INTERFACE I_Telescope

PROPERTY Altitude : LREAL
GET
END_GET
END_PROPERTY

PROPERTY Azimuth : LREAL
GET
END_GET
END_PROPERTY

PROPERTY CoverAutoOpen : BOOL
GET
END_GET
SET
END_SET
END_PROPERTY

PROPERTY Declination : LREAL
GET
END_GET
END_PROPERTY

METHOD ABSTRACT Home : BOOL
VAR_INPUT
END_VAR
END_METHOD

METHOD Init : BOOL
VAR_INPUT
END_VAR
END_METHOD

METHOD ABSTRACT Park : BOOL
VAR_INPUT
END_VAR
END_METHOD

METHOD Reset : BOOL
VAR_INPUT
END_VAR
END_METHOD

PROPERTY RightAscension : LREAL
GET
END_GET
END_PROPERTY

METHOD Slew : BOOL
VAR_INPUT
	fAzimuth		: LREAL;
	fAltitude		: LREAL;
END_VAR
END_METHOD

METHOD Stop : BOOL
VAR_INPUT
END_VAR
END_METHOD

METHOD Track : BOOL
VAR_INPUT
	fRightAscension	: LREAL;
	fDeclination	: LREAL;
END_VAR
END_METHOD

END_INTERFACE

(* stored: Version 1.1.0.1, ProductVersion 3.1.4024.15
   Itf I_Telescope: Id {5003d6e3-4b52-4cb8-a028-b0ab2a6b3370}
   Property Altitude: Id {ce60f76f-3a5f-482f-9275-0897e7d29930}
   Get Get: Id {58c7dbd3-1bf7-4cb4-96b8-f33be68a1ee1}
   Property Azimuth: Id {32bf6858-c17f-4c7b-8e70-4ffdf9df410d}
   Get Get: Id {63e5582f-b70a-403e-801b-c0e6f9154192}
   Property CoverAutoOpen: Id {f8160a73-8302-45f4-9c7c-d48b30d350e4}
   Get Get: Id {d18e5bdf-2192-4bf0-9513-4be35621818a}
   Set Set: Id {292bc5f3-fb7f-4633-b013-091fb338acaf}
   Property Declination: Id {a5cf9f3f-1ec9-4cca-8bd9-8121481b9a9f}
   Get Get: Id {fcb6c1b5-27f0-4565-aed9-45fc0ce88d7e}
   Method Home: Id {2fc689c7-e332-49bc-87f2-069b41e58195}
   Method Init: Id {a446f50b-d891-42c3-bcd4-e100ad4f506e}
   Method Park: Id {4989c55f-52d0-4389-8fa2-916073e653f8}
   Method Reset: Id {7c6108fb-54b5-48bf-af67-cc7170330ed5}
   Property RightAscension: Id {0971e0b4-9db1-4a87-a57f-319f62ce77d0}
   Get Get: Id {137c7751-8023-4049-92ca-329be45aaf37}
   Method Slew: Id {cc0d567e-4a90-40d9-8f8e-e1a94eb43aa2}
   Method Stop: Id {078c3ad2-bc5e-4ad8-9b03-f137aaad29d9}
   Method Track: Id {17caa4eb-aef5-4541-b247-843b6eb5de40} *)
